FUNCTION_BLOCK RT_Bridge_11 (* Data connection decoupling bridge for data connection between real-time event chains *)
  (* Standard: 61499-2; Description: Copyright (c) 2023 Johannes Kepler University Linz This program and the accompanying materials are made available under the terms of the Eclipse Public License 2.0 which is available at https://www.eclipse.org/legal/epl-2.0/ SPDX-License-Identifier: EPL-2.0 *)
  (* Version 1.0, 2023-11-02, Alois Zoitl, Johannes Kepler University Linz *)
  {SET_ATTRIBUTE(GenericClassName, 'GEN_RT_Bridge')}
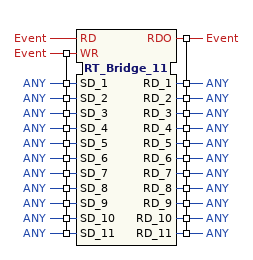
  EVENT_INPUT
    RD; (* Read data from data bridge *)
    WR WITH SD_1, SD_2, SD_3, SD_4, SD_5, SD_6, SD_7, SD_8, SD_9, SD_10, SD_11; (* Write data to data bridge *)
  END_EVENT
  EVENT_OUTPUT
    RDO WITH RD_1, RD_2, RD_3, RD_4, RD_5, RD_6, RD_7, RD_8, RD_9, RD_10, RD_11; (* Read data notifcation *)
  END_EVENT
  VAR_INPUT
    SD_1 : ANY; (* Data to be put into the data bridge *)
    SD_2 : ANY; (* Data to be put into the data bridge *)
    SD_3 : ANY; (* Data to be put into the data bridge *)
    SD_4 : ANY; (* Data to be put into the data bridge *)
    SD_5 : ANY; (* Data to be put into the data bridge *)
    SD_6 : ANY; (* Data to be put into the data bridge *)
    SD_7 : ANY; (* Data to be put into the data bridge *)
    SD_8 : ANY; (* Data to be put into the data bridge *)
    SD_9 : ANY; (* Data to be put into the data bridge *)
    SD_10 : ANY; (* Data to be put into the data bridge *)
    SD_11 : ANY; (* Data to be put into the data bridge *)
  END_VAR
  VAR_OUTPUT
    RD_1 : ANY; (* Data from data bridge *)
    RD_2 : ANY; (* Data from data bridge *)
    RD_3 : ANY; (* Data from data bridge *)
    RD_4 : ANY; (* Data from data bridge *)
    RD_5 : ANY; (* Data from data bridge *)
    RD_6 : ANY; (* Data from data bridge *)
    RD_7 : ANY; (* Data from data bridge *)
    RD_8 : ANY; (* Data from data bridge *)
    RD_9 : ANY; (* Data from data bridge *)
    RD_10 : ANY; (* Data from data bridge *)
    RD_11 : ANY; (* Data from data bridge *)
  END_VAR
  (* Service APPLICATION/RESOURCE: Data connection decoupling bridge for data connection between real-time event chains *)
END_FUNCTION_BLOCK
